// SIMATIC STEP 7 (V5.x) project S_cortar
// station: P_ADR_BUS
// station: Hardware
// station: Equipo SIMATIC 300

SYMBOL_TABLE
"CORTAR"	FC 1	FC 1	// Funcion de cortar las planchas
"bit_de_trabajo"	I 124.0	BOOL
"sensorabajo"	I 124.1	BOOL
"sensorarriba"	I 124.2	BOOL
"expulsada"	I 124.3	BOOL
"OK"	I 124.4	BOOL
"START"	I 124.5	BOOL
"Cycle Execution"	OB 1	OB 1
"bajarcuchilla"	Q 100.0	BOOL
"expulsarplancha"	Q 100.1	BOOL
"bit_ok"	Q 100.2	BOOL
"STBY"	Q 100.3	BOOL
END_SYMBOL_TABLE

FUNCTION "CORTAR" : VOID	// FC 1
TITLE = CORTAR
VERSION : 0.1
VAR_INPUT
  bit_de_trabajo : BOOL ;
  SENSORABAJO : BOOL ;
  SENSORARRIBA : BOOL ;
  EXPULSADA : BOOL ;
  START : BOOL ;
  OK : BOOL ;
END_VAR
VAR_OUTPUT
  BAJARCUCHILLA : BOOL ;
  EXPULSARPLANCHA : BOOL ;
  bit_ok : BOOL ;
  STBY : BOOL ;
END_VAR
VAR_TEMP
  x51 : BOOL ;
  x52 : BOOL ;
  x53 : BOOL ;
  s3 : BOOL ;
  FP_BDT : BOOL ;
  X50 : BOOL ;
  FP_START : BOOL ;
END_VAR
BEGIN
NETWORK
TITLE = Arranque
      A     #bit_de_trabajo;
      FP    #FP_BDT;
      S     #X50;
      R     #x51;
      R     #x52;
      R     #x53;
      R     #s3;
NETWORK
TITLE = de x51 a x52
      A     #x51;
      A     #SENSORABAJO;
      R     #x51;
      S     #x52;
NETWORK
TITLE = de x52 a x53
      A     #x52;
      A     #SENSORARRIBA;
      R     #x52;
      S     #x53;
NETWORK
TITLE = de x53 a s3
      A     #x53;
      A     #EXPULSADA;
      R     #x53;
      S     #s3;
NETWORK
TITLE = Accion x51
      A     #x51;
      =     #BAJARCUCHILLA;
NETWORK
TITLE = Accion x53
      A     #x53;
      =     #EXPULSARPLANCHA;
NETWORK
TITLE = Accion final
      A     #s3;
      =     #bit_ok;
NETWORK
TITLE =
      A     #s3;
      A     #OK;
      R     #s3;
      S     #X50;
NETWORK
TITLE =
      A     #X50;
      A     #START;
      FP    #FP_START;
      R     #X50;
      S     #x51;
NETWORK
TITLE =
      A     #X50;
      =     #STBY;
END_FUNCTION

ORGANIZATION_BLOCK "Cycle Execution"	// OB 1
TITLE = "Main Program Sweep (Cycle)"
VERSION : 0.1
VAR_TEMP
  OB1_EV_CLASS : BYTE ;	//Bits 0-3 = 1 (Coming event), Bits 4-7 = 1 (Event class 1)
  OB1_SCAN_1 : BYTE ;	//1 (Cold restart scan 1 of OB 1), 3 (Scan 2-n of OB 1)
  OB1_PRIORITY : BYTE ;	//Priority of OB Execution
  OB1_OB_NUMBR : BYTE ;	//1 (Organization block 1, OB1)
  OB1_RESERVED_1 : BYTE ;	//Reserved for system
  OB1_RESERVED_2 : BYTE ;	//Reserved for system
  OB1_PREV_CYCLE : INT ;	//Cycle time of previous OB1 scan (milliseconds)
  OB1_MIN_CYCLE : INT ;	//Minimum cycle time of OB1 (milliseconds)
  OB1_MAX_CYCLE : INT ;	//Maximum cycle time of OB1 (milliseconds)
  OB1_DATE_TIME : DATE_AND_TIME ;	//Date and time OB1 started
END_VAR
BEGIN
NETWORK
TITLE =
      CALL  "CORTAR" (
           bit_de_trabajo           := "bit_de_trabajo",
           SENSORABAJO              := "sensorabajo",
           SENSORARRIBA             := "sensorarriba",
           EXPULSADA                := "expulsada",
           START                    := "START",
           OK                       := "OK",
           BAJARCUCHILLA            := "bajarcuchilla",
           EXPULSARPLANCHA          := "expulsarplancha",
           bit_ok                   := "bit_ok",
           STBY                     := "STBY");
END_ORGANIZATION_BLOCK
